TYPE DUT_HMI_UPSStatus :
STRUCT
	Valid : BOOL;
	State : ST_UPSStatus;
END_STRUCT
END_TYPE

(* stored: Version 1.1.0.1, ProductVersion 3.1.4024.13
   DUT DUT_HMI_UPSStatus: Id {b3a8aaa4-c554-4125-9c32-ae9f6db76c0f} *)
